Yaskawa INFORM job: KRIS7_V2.JBI

/JOB
//NAME KRIS7_V2
//POS
///NPOS 420,420,420,15,0,0
///TOOL 0
///POSTYPE PULSE
///PULSE
C00000=4302,-119221,-120806,-3568,29214,482
C00001=4302,-119221,-120806,-3568,29214,482
C00002=-36471,-76527,-106813,19264,71481,77238
C00003=-63812,-119516,-80644,-27282,71106,59809
C00004=-86670,-29465,-24103,-33182,93398,46515
C00005=-88663,-31189,-25266,-33292,92471,45985
C00006=-89600,-31952,-25776,-33339,92036,45737
C00007=-88663,-31189,-25266,-33292,92471,45985
C00008=-88663,-31929,-28188,-33361,93666,45629
C00009=-101397,-33118,-34088,-22474,91022,41668
C00010=-101397,-32934,-33069,-22469,90527,41762
C00011=-101397,-33275,-35023,-22483,91481,41581
C00012=-104499,20623,14787,-23283,115207,62973
C00013=-104352,17765,12486,-23220,115200,63034
C00014=-104529,15851,10717,-23303,115245,62949
C00015=-104352,17765,12486,-23220,115200,63034
C00016=-100086,19810,13187,-22516,115799,63398
C00017=-93288,781,-1160,-33549,91987,44264
C00018=-95103,1586,-482,-33591,91265,43744
C00019=-95638,1156,-842,-33600,91054,43591
C00020=-95103,1586,-482,-33591,91265,43744
C00021=-100253,-3614,-11898,-25466,91372,41970
C00022=-107199,-8537,-17665,-19004,89460,40114
C00023=-108350,-8919,-17473,-17740,88760,39873
C00024=-102096,-5783,-13006,-25389,90415,41488
C00025=-93175,-13453,-24658,-25770,96080,43586
C00026=-29596,-126908,-80456,-16683,91164,67663
C00027=-130966,-130992,-81417,14801,93022,-34731
C00028=-139735,-123676,-71676,23223,79574,-40827
C00029=-136755,-124231,-71804,23689,78586,-39979
C00030=-134984,-124514,-71869,23951,78010,-39473
C00031=-136755,-124231,-71804,23689,78586,-39979
C00032=-136306,-124758,-74432,23664,79703,-39597
C00033=-105195,-127447,-79852,15126,73259,-28242
C00034=-104798,-126140,-77647,15190,72530,-28198
C00035=-108375,-128078,-79564,15067,73342,-29336
C00036=-112121,-93277,-65445,16297,96104,-47809
C00037=-116095,-84503,-58814,18813,102506,-48434
C00038=-114391,-86924,-59797,19239,101506,-47972
C00039=-116095,-84503,-58814,18813,102506,-48434
C00040=-117812,-129995,-81150,14641,74986,-32390
C00041=-118791,-92886,-67151,14205,85296,-31516
C00042=-116748,-92781,-67110,14299,84968,-30842
C00043=-115499,-92681,-67072,14351,84774,-30431
C00044=-116748,-92781,-67110,14299,84968,-30842
C00045=-116748,-94243,-70296,14285,86141,-30707
C00046=-102870,-92009,-70676,9222,86435,-25689
C00047=-102870,-90997,-68303,9229,85506,-25758
C00048=-102870,-92009,-70676,9222,86435,-25689
C00049=-124106,-98193,-79828,8318,91183,-32632
C00050=-120990,-117719,-86799,1028,78019,83969
C00051=-103618,-122878,-84450,6731,45671,69045
C00052=-107839,-39273,-43881,11021,86771,60654
C00053=-102663,-26959,-34255,5037,90909,61236
C00054=-106417,-22492,-30421,10624,98396,60708
C00055=-103076,-37240,-40581,8849,97261,61678
C00056=-110992,-39766,-43585,17340,97602,59383
C00057=-111851,-103912,-94699,10334,87868,68255
C00058=-100525,-93554,-87313,9422,87254,72087
C00059=-95765,-72558,-76889,7644,100510,59309
C00060=-95463,-76426,-71939,16938,115118,61391
C00061=-102124,-64154,-61473,23072,122501,60539
C00062=-108072,-63754,-61449,27079,123073,58329
C00063=-126453,-110744,-88068,25157,96958,85114
C00064=-124535,-114305,-86499,25277,93833,85163
C00065=-121951,-112497,-85625,25654,93398,86032
C00066=-116232,-108405,-84002,26384,92604,88006
C00067=-122754,-106725,-87203,25770,97209,86568
C00068=-142865,-91008,-85242,17891,113758,73123
C00069=-142005,-90205,-84914,18160,113770,73464
C00070=-93871,-48257,-54590,-14207,101968,-48555
C00071=-106716,17042,-5346,-15024,102835,-53222
C00072=-114740,-14345,-34597,-13608,101053,-59815
C00073=-127078,-3386,-21930,-8482,103399,-53955
C00074=-129021,-1243,-17298,-7607,102543,-53064
C00075=-129893,-13096,-22178,-14005,113849,-54571
C00076=-129597,-5294,-13720,-15224,118044,-55057
C00077=-122058,-3228,-13278,-23261,119236,-52777
C00078=-102997,28917,14853,-20600,116287,-84527
C00079=-102792,-6395,-13177,-23260,105514,-87254
C00080=-105472,-3384,-9862,-23514,105257,-88219
C00081=-107060,-2107,-8876,-23770,104848,-88744
C00082=-104416,1445,-8009,-23523,106791,-88129
C00083=-100743,5943,-9423,-11985,113108,-51981
C00084=-104100,-22795,-28366,-25068,61310,-50210
C00085=-122112,-33809,-21710,-17217,45375,-58941
C00086=-130767,-31374,-20493,-827,48037,-55558
C00087=-127443,-25046,-15801,-6227,47707,-53970
C00088=-124818,-6385,-1356,-9028,48013,-52772
C00089=-117469,-7945,-6130,-22808,51414,-49873
C00090=-27812,-119319,-87277,-42007,83182,-24370
C00091=-5621,-139291,-109992,-39952,96377,80222
C00092=-5621,-139291,-109992,-39952,96377,80222
C00093=87039,-115654,-82424,8022,52039,63522
C00094=129513,-144814,-136934,9080,53426,64546
C00095=129513,-144814,-136934,9080,53426,64546
C00096=129513,-109632,-69732,14359,30578,61412
C00097=129513,-83278,-28536,22379,19314,57484
C00098=122399,-55102,-4999,-8402,35911,61097
C00099=119920,-45288,5620,-7331,30390,60229
C00100=119750,-46058,4611,-7150,30605,60108
C00101=119750,-45110,6218,-7257,30106,60163
C00102=119736,-46268,4531,-7151,30546,60106
C00103=119736,-47979,3777,-7238,30135,60151
C00104=119727,-46869,5444,-7329,29678,60198
C00105=119739,-46062,5830,-7299,29854,60181
C00106=119715,-47768,4014,-7231,30094,60141
C00107=122330,-55612,-6297,-8657,32618,61353
C00108=121709,-73745,-24049,9098,30676,53116
C00109=129398,-114812,-46545,3278,22913,57364
C00110=129398,-114812,-46545,3278,22913,57364
C00111=147189,-126166,-80752,5474,34460,60082
C00112=165214,-137669,-115409,7698,46160,62836
C00113=176409,-144814,-136934,9080,53426,64546
C00114=176409,-109327,-69248,14418,30440,61382
C00115=137996,-109327,-69248,14418,30440,61382
C00116=136854,5077,41656,21727,21645,57624
C00117=123203,14789,51546,53172,38991,40073
C00118=123077,34948,78392,59944,35543,36223
C00119=123077,37993,83408,61838,34770,35183
C00120=123098,35348,79007,60153,35442,36112
C00121=123139,31348,74887,59568,35673,36443
C00122=123149,34907,80133,61289,34946,35499
C00123=123130,37074,82445,61677,34805,35280
C00124=123183,30422,73312,58971,35912,36781
C00125=123599,57381,99984,51632,43856,40437
C00126=128629,59731,102899,52063,41097,41453
C00127=130023,30320,69348,52154,35987,38987
C00128=132104,19481,50493,23737,37003,47692
C00129=136200,48792,78585,9333,46433,53780
C00130=127667,43842,73216,11867,48213,50363
C00131=127110,36942,61073,12684,52130,50324
C00132=125174,17943,48073,21449,38985,45601
C00133=109988,7135,45797,56276,48109,34557
C00134=110783,-2370,26113,10588,43916,42309
C00135=96618,15106,36280,16308,48845,36588
C00136=99195,57631,83562,8929,54990,39222
C00137=83229,75338,108095,18392,45531,30732
C00138=82057,52050,70954,17595,54461,31693
C00139=99279,-29834,2408,12633,51480,38376
C00140=124602,-34297,-476,3581,48489,48797
C00141=129000,-155474,-110821,1722,53982,50766
C00142=129000,-186332,-136923,1718,54189,50769
C00143=129000,-186332,-136923,1718,54189,50769
C00144=124634,-42983,-17396,3288,54424,49011
C00145=119975,43106,65207,5416,48088,46799
C00146=124227,21838,45287,-4126,60993,49348
C00147=115102,22260,45694,-2630,60591,46004
C00148=111900,23179,46586,-2094,60423,44829
C00149=106599,25422,48781,-1196,60121,42879
C00150=109500,51617,73450,-2873,46958,44240
C00151=119708,-19564,1692,5024,54962,47046
C00152=124398,4257,31803,38326,49723,41965
C00153=124500,-5455,16693,36249,53145,43496
C00154=123978,22175,41893,32824,63757,46964
C00155=136633,26599,46213,31259,58773,50852
C00156=137127,47274,64261,33367,46328,47205
C00157=127043,-60461,-47717,31537,61680,47716
C00158=130427,-104246,-66216,34447,50964,45598
C00159=130427,-131180,-133049,27346,74705,52630
C00160=129293,-131648,-133187,27764,74930,52255
C00161=129293,-112975,-80869,32941,55210,46617
C00162=125224,-26758,-13299,33226,59088,46051
C00163=97492,-17863,6740,47317,62068,35221
C00164=76763,21057,43225,48272,71101,29312
C00165=80709,51150,75439,39481,73131,33496
C00166=101893,22474,45257,39781,66883,40263
C00167=98002,-1326,18556,46821,62661,35806
C00168=97492,-17863,6740,47317,62068,35221
C00169=125224,-26758,-13299,33226,59088,46051
C00170=129293,-131648,-133187,27764,74930,52255
C00171=129293,-130373,-135142,27565,76585,52657
C00172=129293,-130373,-135142,27565,76585,52657
C00173=129293,-130373,-135142,27565,76585,52657
C00174=126775,-65943,-41926,33631,56357,45828
C00175=146499,-5820,8509,-12483,47348,74367
C00176=133227,18598,33392,-5127,43166,68552
C00177=134087,40556,59352,-4333,44134,68757
C00178=109518,39473,58200,8432,44907,57480
C00179=110804,22133,33080,8574,45677,58038
C00180=95832,-100308,-60228,18401,42759,50383
C00181=85717,-180836,-128237,23276,45701,46095
C00182=134324,-194207,-130804,-6935,34984,69726
C00183=134324,-194207,-130804,-6935,34984,69726
C00184=134324,-194207,-130804,-6935,34984,69726
C00185=126554,-62104,-55568,-768,56192,65237
C00186=102691,-29899,-32559,11070,60126,55987
C00187=93699,-1684,15739,18283,46963,50224
C00188=95177,34388,59282,20423,38809,49091
C00189=95427,37375,44105,11480,58003,52927
C00190=82804,57701,66332,15963,56969,47713
C00191=80078,42075,52490,24500,50349,44630
C00192=92595,-4722,8571,18053,49920,50291
C00193=90890,13188,28851,45241,66990,53478
C00194=96516,51970,78121,48970,56932,51018
C00195=108766,35550,55769,36284,51974,56943
C00196=109501,48300,76470,39344,46724,54946
C00197=112089,47430,75488,38680,45769,55875
C00198=109461,35195,57508,36711,50675,56747
C00199=102961,43860,64049,37370,53600,54832
C00200=117347,37004,56694,33344,48695,60037
C00201=107165,27849,47408,45061,56134,56400
C00202=93699,-1684,15739,18283,46963,50224
C00203=126554,-62104,-55568,-768,56192,65237
C00204=132741,-190295,-136907,-5065,40605,68463
C00205=132741,-190295,-136907,-5065,40605,68463
C00206=132741,-190295,-136907,-5065,40605,68463
C00207=132741,-190295,-136907,-5065,40605,68463
C00208=126216,-48827,-32555,-652,48851,65144
C00209=116157,12397,26645,-836,43828,61032
C00210=107201,15073,29086,4732,43915,56787
C00211=108708,45240,59560,984,53519,57995
C00212=105889,47117,61614,1966,53270,56850
C00213=104117,15965,27840,6481,45345,55424
C00214=116157,12397,26645,-836,43828,61032
C00215=115184,32776,48658,-853,48273,60616
C00216=102009,39914,56094,5283,47719,54846
C00217=104295,38849,56164,-3583,45498,56420
C00218=106773,10666,21679,-1556,45201,57174
C00219=121513,8451,23347,32656,44981,60126
C00220=121479,33249,54130,32703,45073,60132
C00221=136244,38436,59676,26271,39414,66032
C00222=133358,13884,30500,26959,39421,64637
C00223=126216,-48827,-32555,-652,48851,65144
C00224=132741,-190295,-136907,-5065,40605,68463
C00225=132741,-190295,-136907,-5065,40605,68463
C00226=132741,-190295,-136907,-5065,40605,68463
C00227=132741,-190295,-136907,-5065,40605,68463
C00228=126554,-62104,-55568,-768,56192,65237
C00229=93699,-1684,15739,18283,46963,50224
C00230=109219,22842,33799,17593,55341,60017
C00231=114933,32716,55729,7970,41115,61622
C00232=98115,43367,67193,11592,40390,54327
C00233=92675,33947,50979,20393,49569,52577
C00234=113935,26100,44118,24451,47496,60162
C00235=114558,35388,59860,26260,42851,59091
C00236=117732,34768,59212,24806,41998,60459
C00237=114305,24559,43264,24398,47147,60243
C00238=99844,11402,27037,25299,53213,55440
C00239=126554,-62104,-55568,-768,56192,65237
C00240=132741,-190295,-136907,-5065,40605,68463
C00241=132741,-190295,-136907,-5065,40605,68463
C00242=132741,-190295,-136907,-5065,40605,68463
C00243=132741,-190295,-136907,-5065,40605,68463
C00244=126216,-48827,-32555,-652,48851,65144
C00245=134748,7082,18366,-200,46227,68791
C00246=132038,36511,51354,2924,49864,67481
C00247=110399,36003,50767,11764,51912,58463
C00248=101806,27679,40045,16592,51225,54569
C00249=102258,33237,49963,17192,48019,54198
C00250=104874,31614,48575,4374,45128,56525
C00251=106858,16986,29459,6761,48587,57166
C00252=113156,-2573,6178,11839,50347,59373
C00253=100847,-116604,-69788,21646,41420,51852
C00254=93537,-194381,-130385,26473,40988,47897
C00255=64846,-189571,-124664,-20885,48631,75512
C00256=85742,-187574,-126898,-2819,30744,64627
C00257=124193,-185785,-128899,13362,14722,54877
C00258=104459,-185785,-128899,13362,14722,54877
C00259=137185,-168918,-120422,-22616,31853,56508
C00260=103466,-143035,-89833,18127,44217,-664
C00261=153034,-42791,-3789,-574,51224,21077
C00262=154411,-23786,22188,6392,45845,11810
C00263=163692,-14831,30793,3045,43978,15753
C00264=162658,-12144,32796,3380,44162,15317
C00265=162658,-10372,35929,3443,43146,15280
C00266=162658,-10822,35136,3427,43403,15291
C00267=163644,-13399,33193,3102,43239,15709
C00268=163644,-12612,34572,3127,42795,15690
C00269=163043,-11060,35746,3327,42891,15434
C00270=163515,-12286,34819,3170,42815,15635
C00271=166152,-32133,5550,1997,50546,16952
C00272=100006,-46830,-3879,17345,57754,-8477
C00273=55652,-4276,24712,7053,56203,-22524
C00274=50070,19037,58848,16400,45172,-27179
C00275=51341,29328,71603,16783,42484,-27133
C00276=51341,32600,77102,17341,40853,-27469
C00277=51341,31422,75137,17137,41430,-27347
C00278=50264,28853,72458,17349,41942,-27728
C00279=50264,30492,75208,17635,41129,-27900
C00280=50738,31631,76404,17545,40896,-27733
C00281=50419,30858,75590,17605,41054,-27844
C00282=50419,14018,45638,14959,50461,-26136
C00283=53903,-12653,21571,13778,50962,-24612
C00284=66094,-67687,-18476,10677,45688,-20127
C00285=87454,-109874,-47340,-27972,40441,7116
C00286=78946,-55292,-6224,-23492,40558,2756
C00287=70027,-40972,10385,-20890,35738,-464
C00288=63439,-31094,22495,-18522,32104,-3061
C00289=63439,-29243,25592,-19018,31198,-2801
C00290=75556,-28394,37292,-62320,27769,16956
C00291=74155,-27422,37887,-61985,27131,16453
C00292=64318,-30449,24372,-21159,31089,-1672
C00293=67917,-25293,27676,-22824,32488,-51
C00294=67917,-25293,27676,-22824,32488,-51
C00295=68696,-24050,28500,-23162,32795,289
C00296=67917,-25293,27676,-22824,32488,-51
C00297=75368,-51805,-10970,-21451,43738,562
C00298=86139,-25078,5298,-24076,50017,4008
C00299=83917,-18337,16451,-24570,46284,3982
C00300=79836,-11066,25880,-23931,43276,2865
C00301=79836,-9413,28995,-24399,42297,3151
C00302=86314,-11086,32289,-42271,40319,10375
C00303=84998,-9998,33124,-41890,39785,9892
C00304=80963,-11349,26642,-26884,42529,4054
C00305=82363,-6834,30155,-27320,43093,4575
C00306=82761,-5465,31244,-27447,43243,4725
C00307=83186,-3958,32457,-27584,43396,4888
C00308=82761,-5465,31244,-27447,43243,4725
C00309=87385,-23200,183,-25112,53654,3858
C00310=88611,-6659,17671,-26227,51974,4862
C00311=85936,239,26154,-25964,49655,4281
C00312=85936,1480,28752,-26325,48787,4530
C00313=91127,630,32748,-40408,46738,9768
C00314=90313,1326,33333,-40211,46382,9497
C00315=86792,7,26768,-28149,49107,5083
C00316=90602,-33059,-4237,-28517,52203,5912
C00317=94576,-67258,-23025,57506,77870,-531
C00318=122383,-58832,-3556,65417,58097,774
C00319=127343,-13643,25366,63114,57669,4189
C00320=131296,13324,53885,65824,53660,3026
C00321=131296,14618,56173,66322,53341,2642
C00322=130824,14275,55697,67245,54004,2465
C00323=131723,14569,55971,67399,53464,2593
C00324=130860,14268,55674,67244,53987,2476
C00325=127124,-5804,29633,63377,58737,4694
C00326=126701,-15037,22522,63119,61223,3769
C00327=126701,1136,51385,68187,57095,-774
C00328=131284,6353,59362,70779,53649,-1335
C00329=131284,8754,63319,71617,53230,-1977
C00330=131284,6353,59362,70779,53649,-1335
C00331=132452,6685,59657,71098,52984,-1198
C00332=131284,6353,59362,70779,53649,-1335
C00333=131052,11501,64001,70861,53706,-1474
C00334=130893,14100,66417,70922,53742,-1574
C00335=130719,17099,69269,71021,53763,-1708
C00336=130893,14100,66417,70922,53742,-1574
C00337=128315,-22064,27147,66784,57381,941
C00338=129627,-37207,17556,68184,55855,186
C00339=130148,-23471,44300,74760,52317,-4741
C00340=135320,-14449,56479,79067,48853,-5949
C00341=135320,-12066,60154,79963,48630,-6563
C00342=135320,-14449,56479,79067,48853,-5949
C00343=137070,-14043,56767,79770,47945,-5809
C00344=135320,-14449,56479,79067,48853,-5949
C00345=134716,-10676,59212,78597,49226,-5841
C00346=134466,-8976,60486,78417,49378,-5807
C00347=134182,-6930,62050,78227,49545,-5776
C00348=134466,-8976,60486,78417,49378,-5807
C00349=106496,-51026,-9475,59829,73743,881
C00350=106496,-62277,-31108,58328,77765,3910
C00351=137468,-45448,-13164,23993,62707,9546
C00352=142031,-34381,-3630,18745,59946,9254
C00353=153480,-23481,18954,7895,48240,10284
C00354=154576,-15419,32985,7624,43640,10304
C00355=154522,-15140,33190,7639,43662,10282
C00356=163868,-10589,37972,6252,39486,12143
C00357=163705,-4288,45034,21073,38117,2051
C00358=163923,-2936,48273,26703,35302,170
C00359=146970,-27557,19782,29282,44621,-5055
C00360=77984,-28544,12598,9594,52255,-4511
C00361=87028,-14899,33509,-8097,43242,2023
C00362=86974,-14913,33498,-8080,43236,2001
C00363=77485,-7266,39372,-4959,42873,-2067
C00364=74579,-2521,47308,-17915,35684,548
C00365=75615,102,52227,-26296,32839,3633
C00366=84696,-19604,28451,-27180,39406,6073
C00367=87454,-109874,-47340,-27972,40441,7116
C00368=87454,-109874,-47340,-27972,40441,7116
C00369=73980,-36973,3355,-18473,60366,27525
C00370=58877,-27993,19766,-16405,50257,19650
C00371=71120,-6285,35203,-17245,53240,22132
C00372=69479,-8808,33067,-14788,50723,16894
C00373=73605,-31096,1389,-14177,59206,17320
C00374=72431,-18207,17991,-16956,51529,14828
C00375=73562,-15726,19761,-17396,52120,15565
C00376=83313,14185,44247,-21039,56473,22237
C00377=84211,-11070,13701,-18734,53182,26231
C00378=82998,-523,24465,-18637,51768,25979
C00379=82448,-570,28041,-15362,40529,26924
C00380=77134,-2165,39833,11119,14146,19838
C00381=76844,-12553,31864,7458,12108,20601
C00382=84341,-54767,463,-16268,10060,32559
C00383=79893,-46463,9240,-49361,8484,37720
C00384=71243,-22477,30789,30336,5200,-490
C00385=70979,-19028,33557,31433,5346,-1026
C00386=68683,-10375,50772,112552,4351,-37626
C00387=72976,-34040,25530,30096,2440,-170
C00388=51638,-47354,18402,88201,13764,-30312
C00389=50365,-30767,37744,101133,14655,-36527
C00390=46532,-17600,60099,119714,18815,-46088
C00391=50533,-52861,21550,106572,14840,-38992
C00392=66288,-93178,-46103,5866,60369,16168
C00393=112510,-98188,-44790,18471,62864,-44268
C00394=149625,-37879,6780,17046,57011,-35751
C00395=155605,-32525,16928,15112,50177,-29308
C00396=149418,-7594,34122,13784,51545,-27133
C00397=143716,-10385,36525,25765,46016,-27057
C00398=147766,-22217,9496,11268,57983,-23560
C00399=146875,-12758,20894,15319,55227,-24771
C00400=146053,-8471,24161,15451,55560,-25047
C00401=142035,19351,48051,16301,55907,-26583
C00402=141803,14161,44980,18392,51510,-21349
C00403=142040,5818,24378,13474,61789,-22474
C00404=138840,15265,37176,20739,58625,-24937
C00405=138706,17261,38894,20771,58629,-24991
C00406=139526,10572,40705,23596,37058,-29346
C00407=140566,11430,47120,26457,25355,-31911
C00408=140419,-8993,28489,25719,26277,-31573
C00409=142059,-17553,21658,25375,25949,-31323
C00410=143624,-11159,28730,24740,24544,-30775
C00411=144392,-5853,43056,31020,18891,-33660
C00412=150093,-42733,14524,24992,16002,-29807
C00413=146967,-32270,24662,40502,20136,-34953
C00414=144755,-20255,35089,33636,31779,-30408
C00415=144236,-61611,5153,41773,14596,-38681
C00416=136995,-150356,-85047,33892,64386,-36535
C00417=136995,-178339,-110283,33604,8697,-36217
C00418=130728,-161100,-136081,16173,33339,-28558
C00419=1271,-161100,-136081,16173,33339,-28558
BC00000=132383,679261,975760
BC00001=132383,679261,975760
BC00002=295325,674563,1075170
BC00003=396971,731967,797664
BC00004=396971,731967,797664
BC00005=396971,731967,797664
BC00006=396971,731967,797664
BC00007=396971,731967,797664
BC00008=396971,731967,797664
BC00009=396971,731967,797664
BC00010=396971,731967,797664
BC00011=396971,731967,797664
BC00012=396971,731967,797664
BC00013=396971,731967,797664
BC00014=396971,731967,797664
BC00015=396971,731967,797664
BC00016=396971,731967,797664
BC00017=396971,731967,797664
BC00018=396971,731967,797664
BC00019=396971,731967,797664
BC00020=396971,731967,797664
BC00021=396971,731967,797664
BC00022=396971,731967,797664
BC00023=396971,731967,797664
BC00024=396971,731967,797664
BC00025=396971,731967,797664
BC00026=396971,731967,797664
BC00027=1331,731967,797664
BC00028=1331,834817,797664
BC00029=1331,834817,797664
BC00030=1331,834817,797664
BC00031=1331,834817,797664
BC00032=1331,834817,797664
BC00033=1331,834817,797664
BC00034=1331,834817,797664
BC00035=1331,834817,797664
BC00036=1331,834817,797664
BC00037=1331,834817,797664
BC00038=1331,834817,797664
BC00039=1331,834817,797664
BC00040=1331,834817,797664
BC00041=1331,834817,797664
BC00042=1331,834817,797664
BC00043=1331,834817,797664
BC00044=1331,834817,797664
BC00045=1331,834817,797664
BC00046=1331,834817,797664
BC00047=1331,834817,797664
BC00048=1331,834817,797664
BC00049=1331,834817,797664
BC00050=1072,761065,516765
BC00051=1072,827865,516765
BC00052=1071,829671,517043
BC00053=1071,829895,517078
BC00054=1071,829895,517078
BC00055=1071,829895,517078
BC00056=1071,829895,517078
BC00057=768,829895,695080
BC00058=768,829895,695080
BC00059=768,829895,695080
BC00060=768,829895,695080
BC00061=768,829895,695080
BC00062=768,829895,695080
BC00063=768,829895,695080
BC00064=768,829895,695080
BC00065=768,829895,695080
BC00066=768,829895,695080
BC00067=768,829895,695080
BC00068=768,829895,695080
BC00069=768,686767,695080
BC00070=396971,681851,797664
BC00071=396971,731967,797664
BC00072=396971,731967,797664
BC00073=396971,731967,797664
BC00074=396971,731967,797664
BC00075=396971,731967,797664
BC00076=396971,731967,797664
BC00077=396971,731967,797664
BC00078=396971,731967,797664
BC00079=396971,731967,797664
BC00080=396971,731967,797664
BC00081=396971,731967,797664
BC00082=396971,731967,797664
BC00083=396971,731967,797664
BC00084=396971,731967,516765
BC00085=396971,731967,516765
BC00086=396971,731967,516765
BC00087=396972,731979,516765
BC00088=396971,731967,516765
BC00089=396971,731967,516765
BC00090=396971,731967,516765
BC00091=188286,731967,1013423
BC00092=188286,774486,1052805
BC00093=125948,1177450,1071719
BC00094=215453,1309115,984509
BC00095=345399,1357897,984509
BC00096=345399,1357897,984509
BC00097=345399,1230997,984509
BC00098=346767,1230997,984506
BC00099=346767,1230997,984506
BC00100=346767,1230997,984506
BC00101=346767,1230997,984506
BC00102=346767,1230997,984506
BC00103=346767,1230997,984506
BC00104=346767,1230997,984506
BC00105=346767,1230997,984506
BC00106=346767,1230997,984506
BC00107=346767,1230997,984506
BC00108=309515,1253158,984507
BC00109=309515,1253158,984507
BC00110=309515,1328360,1051553
BC00111=314470,1361455,1064018
BC00112=253389,1357693,1050986
BC00113=215453,1309115,984509
BC00114=215453,1309115,984509
BC00115=135997,1309115,984509
BC00116=135997,1309115,984509
BC00117=135997,1309115,984509
BC00118=135997,1309115,984505
BC00119=135997,1309115,984505
BC00120=135997,1309115,984505
BC00121=135997,1309115,984505
BC00122=135997,1309115,984505
BC00123=135997,1309115,984505
BC00124=135997,1309115,984505
BC00125=135997,1309115,984509
BC00126=135997,1309115,984509
BC00127=135997,1309115,984509
BC00128=135997,1309115,984509
BC00129=135997,1309115,984509
BC00130=135997,1309115,984509
BC00131=135997,1309115,984509
BC00132=135997,1309115,984509
BC00133=135997,1309115,984509
BC00134=135997,1309115,984509
BC00135=94463,1309115,955550
BC00136=94463,1309115,963176
BC00137=94463,1309115,963176
BC00138=94463,1309115,963176
BC00139=94463,1309115,963176
BC00140=141941,1309115,963176
BC00141=141941,1309115,963176
BC00142=223116,1330631,963176
BC00143=328548,1330631,963176
BC00144=328548,1330631,963176
BC00145=328548,1330631,963176
BC00146=328548,1285890,963176
BC00147=328548,1285890,963176
BC00148=328548,1285890,963176
BC00149=328548,1285890,963176
BC00150=328548,1330631,963176
BC00151=328548,1291307,959498
BC00152=328548,1293601,963176
BC00153=328548,1288886,905196
BC00154=328548,1288886,905196
BC00155=328548,1288886,905196
BC00156=328824,1330631,905196
BC00157=328824,1330631,905196
BC00158=328824,1330631,905196
BC00159=328824,1330631,905196
BC00160=151003,1330631,905196
BC00161=151003,1330631,905196
BC00162=151003,1330631,905196
BC00163=103648,1289163,905196
BC00164=103648,1289163,905196
BC00165=103648,1289163,905196
BC00166=103648,1289163,905196
BC00167=103648,1289163,905196
BC00168=103648,1289163,905196
BC00169=151003,1330631,905196
BC00170=151003,1330631,905196
BC00171=151003,1330631,905196
BC00172=303803,1330631,905196
BC00173=303803,1330631,763831
BC00174=303803,1330631,902112
BC00175=303803,1330631,902112
BC00176=303803,1330631,902112
BC00177=303803,1330631,902112
BC00178=303803,1330631,902112
BC00179=303803,1330631,902112
BC00180=303803,1330631,902112
BC00181=303803,1330631,1003127
BC00182=236612,1330631,1003127
BC00183=137483,1330631,1003127
BC00184=136337,1325904,719417
BC00185=136337,1325904,818715
BC00186=87820,1325904,842743
BC00187=87820,1325904,951848
BC00188=87820,1325904,951848
BC00189=87820,1320020,844218
BC00190=87820,1320020,844218
BC00191=87820,1325904,927335
BC00192=87820,1325904,927335
BC00193=87820,1325904,927335
BC00194=87820,1325904,927335
BC00195=87820,1325904,927335
BC00196=87820,1325904,927335
BC00197=87820,1325904,927335
BC00198=87820,1325904,927335
BC00199=87820,1325904,890762
BC00200=87820,1325904,890392
BC00201=87820,1325904,927335
BC00202=87820,1325904,951848
BC00203=136337,1325904,818715
BC00204=136337,1325904,818715
BC00205=136337,1325904,998300
BC00206=310720,1325904,998300
BC00207=310720,1325904,777065
BC00208=310720,1325904,891809
BC00209=310720,1325904,891809
BC00210=310720,1325904,891809
BC00211=310720,1325904,891809
BC00212=310720,1325904,891809
BC00213=310720,1325904,891809
BC00214=310720,1325904,891809
BC00215=310720,1325904,891809
BC00216=310720,1325904,891809
BC00217=310720,1325904,891809
BC00218=310720,1325904,891809
BC00219=310720,1325904,891809
BC00220=310720,1325904,891809
BC00221=310720,1325904,891809
BC00222=310720,1325904,891809
BC00223=310720,1325904,891809
BC00224=310720,1325904,777065
BC00225=310720,1325904,998300
BC00226=136337,1325904,998300
BC00227=136337,1325904,818715
BC00228=136337,1325904,818715
BC00229=87820,1325904,951848
BC00230=87820,1325904,927335
BC00231=87820,1325904,927335
BC00232=87820,1325904,927335
BC00233=87820,1325904,927335
BC00234=87820,1325904,927335
BC00235=87820,1325904,927335
BC00236=87820,1325904,927335
BC00237=87820,1325904,927335
BC00238=87820,1325904,927335
BC00239=136337,1325904,818715
BC00240=136337,1325904,818715
BC00241=136337,1325904,998300
BC00242=310720,1325904,998300
BC00243=310720,1325904,777065
BC00244=310720,1325904,891809
BC00245=310720,1325904,891809
BC00246=310720,1325904,891809
BC00247=310720,1325904,891809
BC00248=310720,1325904,891809
BC00249=310720,1325904,891809
BC00250=310720,1325904,891809
BC00251=310720,1325904,891809
BC00252=310720,1325904,891809
BC00253=310720,1325904,891809
BC00254=310720,1325904,1051225
BC00255=156074,1050332,1052018
BC00256=153940,1198656,1051600
BC00257=230237,1331507,1051225
BC00258=230237,1331507,1051225
BC00259=214487,1257960,1051225
BC00260=187930,1133951,1051225
BC00261=187930,1063861,1051225
BC00262=187930,1063861,1051225
BC00263=187931,1063862,1051199
BC00264=187931,1063862,1051199
BC00265=187931,1063862,1051199
BC00266=187931,1063862,1051199
BC00267=187931,1063862,1051199
BC00268=187931,1063862,1051199
BC00269=187931,1063862,1051199
BC00270=187931,1063862,1051199
BC00271=187931,1063862,1051199
BC00272=187930,1063861,1051225
BC00273=187930,1063861,1051225
BC00274=187930,1063861,1051225
BC00275=187930,1063861,1051225
BC00276=187930,1063861,1051225
BC00277=187930,1063861,1051225
BC00278=187930,1063861,1051225
BC00279=187930,1063861,1051225
BC00280=187930,1063861,1051225
BC00281=187930,1063861,1051225
BC00282=187930,1063861,1051225
BC00283=187930,1063861,1051225
BC00284=187930,1063861,1051225
BC00285=244084,1125149,1051225
BC00286=244084,1125149,1051225
BC00287=244084,1125149,1051225
BC00288=244084,1125149,1051225
BC00289=244084,1125149,1051225
BC00290=244084,1125149,1051225
BC00291=244084,1125149,1051225
BC00292=244084,1125149,1051225
BC00293=244084,1125149,1051225
BC00294=244084,1125149,1051225
BC00295=244084,1125149,1051225
BC00296=244084,1125149,1051225
BC00297=244084,1125149,1051225
BC00298=244084,1125149,1051225
BC00299=244084,1125149,1051225
BC00300=244084,1125149,1051225
BC00301=244084,1125149,1051225
BC00302=244084,1125149,1051225
BC00303=244084,1125149,1051225
BC00304=244084,1125149,1051225
BC00305=244084,1125149,1051225
BC00306=244084,1125149,1051225
BC00307=244084,1125149,1051225
BC00308=244084,1125149,1051225
BC00309=244084,1125149,1051225
BC00310=244084,1125149,1051225
BC00311=244083,1125149,1051222
BC00312=244083,1125149,1051222
BC00313=244083,1125149,1051222
BC00314=244083,1125149,1051222
BC00315=244083,1125149,1051222
BC00316=244083,1125149,1051222
BC00317=244083,1125148,1051219
BC00318=166173,1125148,1051219
BC00319=166173,1125148,1051219
BC00320=166173,1142192,1051219
BC00321=166173,1142192,1051219
BC00322=166173,1142192,1051219
BC00323=166173,1142192,1051219
BC00324=166173,1142192,1051219
BC00325=166173,1142192,1051219
BC00326=166173,1142192,1051219
BC00327=166173,1142192,1051219
BC00328=166173,1142192,1051219
BC00329=166173,1142192,1051219
BC00330=166173,1142192,1051219
BC00331=166173,1142192,1051219
BC00332=166173,1142192,1051219
BC00333=166173,1142192,1051219
BC00334=166173,1142192,1051219
BC00335=166173,1142192,1051219
BC00336=166173,1142192,1051219
BC00337=166173,1142192,1051219
BC00338=166173,1142192,1051219
BC00339=166173,1142192,1051219
BC00340=166173,1142192,1051219
BC00341=166173,1142192,1051219
BC00342=166173,1142192,1051219
BC00343=166173,1142192,1051219
BC00344=166173,1142192,1051219
BC00345=166173,1142192,1051219
BC00346=166173,1142192,1051219
BC00347=166173,1142192,1051219
BC00348=166173,1142192,1051219
BC00349=166173,1142192,1051219
BC00350=166173,1142192,1051219
BC00351=180177,1091773,1051223
BC00352=182943,1081815,1051224
BC00353=187709,1064658,1051225
BC00354=187930,1063861,1051225
BC00355=187930,1063861,1051225
BC00356=187930,1063861,1051225
BC00357=187930,1063861,1051225
BC00358=187930,1063861,1051225
BC00359=187930,1063861,1051225
BC00360=244084,1063861,1051225
BC00361=244084,1063861,1051225
BC00362=244084,1063861,1051225
BC00363=244084,1063861,1051225
BC00364=244084,1063861,1051225
BC00365=244084,1063861,1051225
BC00366=244084,1063861,1051225
BC00367=244084,1063861,1051225
BC00368=244084,1125149,1051225
BC00369=244084,1125149,1051225
BC00370=244084,1125149,1051225
BC00371=244084,1125149,1051225
BC00372=244084,1125149,1051225
BC00373=244084,1125149,1051225
BC00374=244084,1125149,1051225
BC00375=244084,1125149,1051225
BC00376=244084,1125149,1051225
BC00377=244084,1125149,1051225
BC00378=244084,1125149,1051225
BC00379=244084,1125149,1051225
BC00380=244084,1125149,1051225
BC00381=244084,1125149,1051225
BC00382=244084,1125149,1051225
BC00383=244084,1125149,1051225
BC00384=244084,1125149,1051225
BC00385=244084,1125149,1051222
BC00386=244084,1125149,1051225
BC00387=244084,1125149,1051225
BC00388=244084,1125149,1051225
BC00389=244083,1125149,1051223
BC00390=244084,1125149,1051225
BC00391=244084,1125149,1051225
BC00392=244084,1125149,1051225
BC00393=148492,1125149,1051225
BC00394=148492,1157650,1055882
BC00395=148492,1157650,1055882
BC00396=148492,1157650,1055882
BC00397=148493,1157650,1055879
BC00398=148492,1157650,1055882
BC00399=148492,1157650,1055882
BC00400=148492,1157650,1055882
BC00401=148492,1157650,1055882
BC00402=148492,1157650,1055882
BC00403=148492,1157650,1055882
BC00404=148492,1157650,1055882
BC00405=148492,1157650,1055882
BC00406=148492,1157650,1055881
BC00407=148492,1157650,1055882
BC00408=148492,1157650,1055882
BC00409=148492,1157650,1055882
BC00410=148492,1157650,1055882
BC00411=148492,1157650,1055882
BC00412=148492,1157650,1055882
BC00413=148492,1157650,1055882
BC00414=148492,1157650,1055882
BC00415=148492,1157650,1055882
BC00416=148492,1157650,1055882
BC00417=189366,1229859,1070827
BC00418=189366,1118575,1070827
BC00419=189366,734808,1070827
EC00000=443420,556475
EC00001=0,556475
EC00002=-88685,-556476
EC00003=-88685,-556476
EC00004=-88685,-556476
EC00005=-88685,-556476
EC00006=-88685,-556476
EC00007=-88685,-556476
EC00008=-88685,-556476
EC00009=-88685,-556476
EC00010=-88685,-556476
EC00011=-88685,-556476
EC00012=-88685,-556476
EC00013=-88685,-556476
EC00014=-88685,-556476
EC00015=-88685,-556476
EC00016=-88685,-556476
EC00017=-88685,-556476
EC00018=-88685,-556476
EC00019=-88685,-556476
EC00020=-88685,-556476
EC00021=-88685,-556476
EC00022=-88685,-556476
EC00023=-88685,-556476
EC00024=-88685,-556476
EC00025=-88685,-556476
EC00026=-88685,-556476
EC00027=-88685,-556476
EC00028=-88685,-556476
EC00029=-88685,-556476
EC00030=-88685,-556476
EC00031=-88685,-556476
EC00032=-88685,-556476
EC00033=-88685,-556476
EC00034=-88685,-556476
EC00035=-88685,-556476
EC00036=-88685,-556476
EC00037=-88685,-556476
EC00038=-88685,-556476
EC00039=-88685,-556476
EC00040=-88685,-556476
EC00041=-88685,-556476
EC00042=-88685,-556476
EC00043=-88685,-556476
EC00044=-88685,-556476
EC00045=-88685,-556476
EC00046=-88685,-556476
EC00047=-88685,-556476
EC00048=-88685,-556476
EC00049=-88685,-556476
EC00050=264893,-556476
EC00051=264893,-556476
EC00052=264346,-556476
EC00053=264278,-556476
EC00054=264278,-556476
EC00055=264278,-556476
EC00056=264278,-556476
EC00057=-85879,-556476
EC00058=-85879,-556476
EC00059=-85879,-556476
EC00060=-85879,-556476
EC00061=-85879,-556476
EC00062=-85879,-556476
EC00063=-85879,-556476
EC00064=-85879,-556476
EC00065=-85879,-556476
EC00066=-85879,-556476
EC00067=-85879,-556476
EC00068=-85879,-556476
EC00069=-85879,-556476
EC00070=-88685,-556476
EC00071=-88685,-556476
EC00072=-88685,-612042
EC00073=-88685,-612042
EC00074=-88685,-612042
EC00075=-88685,-612042
EC00076=-88685,-612042
EC00077=-88685,-612042
EC00078=-88685,-556476
EC00079=-88685,-556476
EC00080=-88685,-556476
EC00081=-88685,-556476
EC00082=-88685,-556476
EC00083=-88685,-556476
EC00084=264893,-556476
EC00085=264893,-605076
EC00086=264893,-605076
EC00087=264894,-605076
EC00088=264893,-605076
EC00089=264893,-605076
EC00090=264893,-556476
EC00091=264890,-556476
EC00092=264890,-556476
EC00093=-210078,-556477
EC00094=-270405,-556477
EC00095=-270405,-556477
EC00096=-270405,-556477
EC00097=-270405,-556477
EC00098=-270404,-556477
EC00099=-270404,-556477
EC00100=-270404,-556477
EC00101=-270404,-556477
EC00102=-270404,-556477
EC00103=-270404,-556477
EC00104=-270404,-556477
EC00105=-270404,-556477
EC00106=-270404,-556477
EC00107=-270404,-556477
EC00108=-270404,-556477
EC00109=-270404,-556477
EC00110=-270404,-556477
EC00111=-270404,-556477
EC00112=-270405,-556477
EC00113=-270405,-556477
EC00114=-270405,-556477
EC00115=-270405,-556477
EC00116=-270405,-556477
EC00117=-270405,-556477
EC00118=-270404,-556477
EC00119=-270404,-556477
EC00120=-270404,-556477
EC00121=-270404,-556477
EC00122=-270404,-556477
EC00123=-270404,-556477
EC00124=-270404,-556477
EC00125=-270405,-556477
EC00126=-270405,-556477
EC00127=-270405,-556477
EC00128=-270405,-556477
EC00129=-270405,-556477
EC00130=-270405,-556477
EC00131=-270405,-556477
EC00132=-270405,-556477
EC00133=-270405,-556477
EC00134=-270405,-556477
EC00135=-270405,-556477
EC00136=-270405,-556477
EC00137=-270405,-556477
EC00138=-270405,-556477
EC00139=-270405,-556477
EC00140=-270405,-556477
EC00141=-270405,-556477
EC00142=-270405,-556477
EC00143=-270405,-556477
EC00144=-270405,-556477
EC00145=-270405,-556477
EC00146=-270405,-556477
EC00147=-270405,-556477
EC00148=-270405,-556477
EC00149=-270405,-556477
EC00150=-270405,-556477
EC00151=-270405,-556477
EC00152=-270405,-556477
EC00153=-270405,-556477
EC00154=-270405,-556477
EC00155=-270405,-556477
EC00156=-270405,-556477
EC00157=-270405,-556477
EC00158=-270405,-556477
EC00159=-270405,-556477
EC00160=-270405,-556477
EC00161=-270405,-556477
EC00162=-270405,-556477
EC00163=-270405,-556477
EC00164=-270405,-556477
EC00165=-270405,-556477
EC00166=-270405,-556477
EC00167=-270405,-556477
EC00168=-270405,-556477
EC00169=-270405,-556477
EC00170=-270405,-556477
EC00171=-270405,-556477
EC00172=-270405,-556477
EC00173=-270405,-556477
EC00174=-270405,-556477
EC00175=-270405,-556477
EC00176=-270405,-556477
EC00177=-270405,-556477
EC00178=-270405,-556477
EC00179=-270405,-556477
EC00180=-270405,-556477
EC00181=-270405,-556477
EC00182=-270405,-556477
EC00183=-270405,-556477
EC00184=-270405,-556477
EC00185=-270405,-556477
EC00186=-270405,-556477
EC00187=-270405,-556477
EC00188=-270405,-556477
EC00189=-270405,-556477
EC00190=-270405,-556477
EC00191=-270405,-556477
EC00192=-270405,-556477
EC00193=-270405,-556477
EC00194=-270405,-556477
EC00195=-270405,-556477
EC00196=-270405,-556477
EC00197=-270405,-556477
EC00198=-270405,-556477
EC00199=-270405,-556477
EC00200=-270405,-556477
EC00201=-270405,-556477
EC00202=-270405,-556477
EC00203=-270405,-556477
EC00204=-270405,-556477
EC00205=-270405,-556477
EC00206=-270405,-556477
EC00207=-270405,-556477
EC00208=-270405,-556477
EC00209=-270405,-556477
EC00210=-270405,-556477
EC00211=-270405,-556477
EC00212=-270405,-556477
EC00213=-270405,-556477
EC00214=-270405,-556477
EC00215=-270405,-556477
EC00216=-270405,-556477
EC00217=-270405,-556477
EC00218=-270405,-556477
EC00219=-270405,-556477
EC00220=-270405,-556477
EC00221=-270405,-556477
EC00222=-270405,-556477
EC00223=-270405,-556477
EC00224=-270405,-556477
EC00225=-270405,-556477
EC00226=-270405,-556477
EC00227=-270405,-556477
EC00228=-270405,-556477
EC00229=-270405,-556477
EC00230=-270405,-556477
EC00231=-270405,-556477
EC00232=-270405,-556477
EC00233=-270405,-556477
EC00234=-270405,-556477
EC00235=-270405,-556477
EC00236=-270405,-556477
EC00237=-270405,-556477
EC00238=-270405,-556477
EC00239=-270405,-556477
EC00240=-270405,-556477
EC00241=-270405,-556477
EC00242=-270405,-556477
EC00243=-270405,-556477
EC00244=-270405,-556477
EC00245=-270405,-556477
EC00246=-270405,-556477
EC00247=-270405,-556477
EC00248=-270405,-556477
EC00249=-270405,-556477
EC00250=-270405,-556477
EC00251=-270405,-556477
EC00252=-270405,-556477
EC00253=-270405,-556477
EC00254=-270405,-556477
EC00255=-1607,-556476
EC00256=-143402,-556477
EC00257=-270405,-556477
EC00258=-270405,-556477
EC00259=-270405,-556477
EC00260=-270405,-556477
EC00261=-270405,-556477
EC00262=-270405,-556477
EC00263=-270402,-556478
EC00264=-270402,-556478
EC00265=-270402,-556478
EC00266=-270402,-556478
EC00267=-270402,-556478
EC00268=-270402,-556478
EC00269=-270402,-556478
EC00270=-270402,-556478
EC00271=-270402,-556478
EC00272=-270405,-556477
EC00273=-270405,-556477
EC00274=-270405,-556477
EC00275=-270405,-556477
EC00276=-270405,-556477
EC00277=-270405,-556477
EC00278=-270405,-556477
EC00279=-270405,-556477
EC00280=-270405,-556477
EC00281=-270405,-556477
EC00282=-270405,-556477
EC00283=-270405,-556477
EC00284=-270405,-556477
EC00285=-447795,-556477
EC00286=-447795,-556477
EC00287=-447795,-556477
EC00288=-447795,-556477
EC00289=-447795,-556477
EC00290=-447795,-556477
EC00291=-447795,-556477
EC00292=-447795,-556477
EC00293=-447795,-556477
EC00294=-447795,-556477
EC00295=-447795,-556477
EC00296=-447795,-556477
EC00297=-447795,-556477
EC00298=-447795,-556477
EC00299=-447795,-556477
EC00300=-447795,-556477
EC00301=-447795,-556477
EC00302=-447795,-556477
EC00303=-447795,-556477
EC00304=-447795,-556477
EC00305=-447795,-556477
EC00306=-447795,-556477
EC00307=-447795,-556477
EC00308=-447795,-556477
EC00309=-447795,-556477
EC00310=-447795,-556477
EC00311=-447793,-556477
EC00312=-447793,-556477
EC00313=-447793,-556477
EC00314=-447793,-556477
EC00315=-447793,-556477
EC00316=-447793,-556477
EC00317=-447791,-556477
EC00318=-447791,-556477
EC00319=-447791,-556477
EC00320=-447791,-556477
EC00321=-447791,-556477
EC00322=-447791,-556477
EC00323=-447791,-556477
EC00324=-447791,-556477
EC00325=-447791,-556477
EC00326=-447791,-556477
EC00327=-447791,-556477
EC00328=-447791,-556477
EC00329=-447791,-556477
EC00330=-447791,-556477
EC00331=-447791,-556477
EC00332=-447791,-556477
EC00333=-447791,-556477
EC00334=-447791,-556477
EC00335=-447791,-556477
EC00336=-447791,-556477
EC00337=-447791,-556477
EC00338=-447791,-556477
EC00339=-447791,-556477
EC00340=-447791,-556477
EC00341=-447791,-556477
EC00342=-447791,-556477
EC00343=-447791,-556477
EC00344=-447791,-556477
EC00345=-447791,-556477
EC00346=-447791,-556477
EC00347=-447791,-556477
EC00348=-447791,-556477
EC00349=-447791,-556477
EC00350=-447791,-556477
EC00351=-333615,-556477
EC00352=-311064,-556477
EC00353=-272209,-556477
EC00354=-270405,-556477
EC00355=-270405,-556477
EC00356=-270405,-556477
EC00357=-270405,-556477
EC00358=-270405,-556477
EC00359=-270405,-556477
EC00360=-270405,-556477
EC00361=-270405,-556477
EC00362=-270405,-556477
EC00363=-270405,-556477
EC00364=-270405,-556477
EC00365=-270405,-556477
EC00366=-270405,-556477
EC00367=-270405,-556477
EC00368=-447795,-556477
EC00369=-447795,-556477
EC00370=-447795,-556477
EC00371=-447795,-556477
EC00372=-447795,-556477
EC00373=-447795,-556477
EC00374=-447795,-556477
EC00375=-447795,-556477
EC00376=-447795,-556477
EC00377=-447795,-556477
EC00378=-447795,-556477
EC00379=-447795,-556477
EC00380=-447795,-556477
EC00381=-447795,-556477
EC00382=-447795,-556477
EC00383=-447795,-556477
EC00384=-447795,-556477
EC00385=-447794,-556477
EC00386=-447795,-556477
EC00387=-447795,-556477
EC00388=-447795,-556477
EC00389=-447794,-556478
EC00390=-447795,-556477
EC00391=-447795,-556477
EC00392=-447795,-556477
EC00393=-447795,-556477
EC00394=-447795,-556477
EC00395=-447795,-556477
EC00396=-447795,-556477
EC00397=-447793,-556477
EC00398=-447795,-556477
EC00399=-447795,-556477
EC00400=-447795,-556477
EC00401=-447795,-556477
EC00402=-447795,-556477
EC00403=-447795,-556477
EC00404=-447795,-556477
EC00405=-447795,-556477
EC00406=-447794,-556478
EC00407=-447795,-556477
EC00408=-447795,-556477
EC00409=-447795,-556477
EC00410=-447795,-556477
EC00411=-447795,-556477
EC00412=-447795,-556477
EC00413=-447795,-556477
EC00414=-447795,-556477
EC00415=-447795,-556477
EC00416=-447795,-556477
EC00417=-447795,-556477
EC00418=-71624,-556477
EC00419=15446,-556477
///POSTYPE BASE
///RECTAN
///RCONF 0,0,0,0,0,0,0,0,0,0,0,0,0,0,0,0,0,0,0,0,0,0,0,0
P00006=0.000,0.000,0.000,0.0000,0.0000,0.0000
P00032=1.957,0.503,-7.217,0.0000,0.0000,0.0000
///RCONF 0,0,0,0,1,0,0,0,0,0,0,0,0,0,0,0,0,0,0,0,0,0,0,0
P00033=-0.123,0.612,-5.012,0.0000,0.0000,0.0000
///RCONF 0,0,0,0,0,0,0,0,0,0,0,0,0,0,0,0,0,0,0,0,0,0,0,0
P00034=-0.304,0.773,-2.693,0.0000,0.0000,0.0000
P00035=2.817,0.591,-1.622,0.0000,0.0000,0.0000
P00040=-0.030,9.648,2.467,0.0000,0.0000,0.0000
P00041=0.192,3.924,0.305,0.0000,0.0000,0.0000
P00042=-0.217,1.941,0.413,0.0000,0.0000,0.0000
P00043=-0.044,-1.937,1.197,0.0000,0.0000,0.0000
P00044=0.687,-2.322,1.156,0.0000,0.0000,0.0000
P00045=-0.068,-0.810,1.603,0.0000,0.0000,0.0000
P00046=0.799,0.043,1.292,0.0000,0.0000,0.0000
P00048=2.411,0.025,-0.606,0.0000,0.0000,0.0000
P00049=3.413,-3.572,-1.618,0.0000,0.0000,0.0000
P00050=4.296,-4.501,-0.826,0.0000,0.0000,0.0000
//INST
///DATE 2025/03/14 12:45
///ATTR SC,RW
///GROUP1 RB1,BS1
///GROUP2 ST1
NOP
MOVJ C00000 BC00000 VJ=100.00  +MOVJ EC00000 VJ=100.00
MOVJ C00001 BC00001 VJ=100.00  +MOVJ EC00001 VJ=100.00
MOVJ C00002 BC00002 VJ=100.00  +MOVJ EC00002 VJ=100.00
CALL JOB:CLEAN-R1_KM_3P
MOVJ C00003 BC00003 VJ=100.00  +MOVJ EC00003 VJ=100.00
MOVJ C00004 BC00004 VJ=50.00  +MOVJ EC00004 VJ=50.00
SMOVL C00005 BC00005 V=83.3  +MOVJ EC00005
SREFP 3 C00006 BC00006  +REFP EC00006
CALL JOB:SEARCH-R1-S13D
SET P032 P006
SFTON3D P032
SMOVL C00007 BC00007 V=60.0  +MOVJ EC00007
SMOVL C00008 BC00008 V=133.3  +MOVJ EC00008
SMOVL C00009 BC00009 V=133.3  +MOVJ EC00009
SREFP 3 C00010 BC00010  +REFP EC00010
CALL JOB:SEARCH-R1-S13D
SET P032 P006
SFTON3D P032
SMOVL C00011 BC00011 V=60.0  +MOVJ EC00011
SMOVL C00012 BC00012 V=133.3  +MOVJ EC00012
SMOVL C00013 BC00013 V=133.3  +MOVJ EC00013
SREFP 3 C00014 BC00014  +REFP EC00014
CALL JOB:SEARCH-R1-S13D
SET P032 P006
SFTON3D P032
SFTOF3D
SMOVL C00015 BC00015 V=133.3  +MOVJ EC00015
SMOVL C00016 BC00016 V=200.0  +MOVJ EC00016
SFTOF3D
'S1
MOVJ C00017 BC00017 VJ=50.00  +MOVJ EC00017 VJ=50.00
'S2
SMOVL C00018 BC00018 V=60.0  +MOVJ EC00018
SREFP 3 C00019 BC00019  +REFP EC00019
CALL JOB:SEARCH-R1-S13D
SET P033 P006
SFTON3D P033
SMOVL C00020 BC00020 V=60.0  +MOVJ EC00020
SMOVL C00021 BC00021 V=133.3  +MOVJ EC00021
SMOVL C00022 BC00022 V=133.3  +MOVJ EC00022
SREFP 3 C00023 BC00023  +REFP EC00023
CALL JOB:SEARCH-R1-S13D
SET P033 P006
SFTON3D P033
SFTOF3D
SMOVL C00024 BC00024 V=83.3  +MOVJ EC00024
MOVJ C00025 BC00025 VJ=60.00  +MOVJ EC00025 VJ=60.00
MOVJ C00026 BC00026 VJ=60.00  +MOVJ EC00026 VJ=60.00
MOVJ C00027 BC00027 VJ=100.00  +MOVJ EC00027 VJ=60.00
MOVJ C00028 BC00028 VJ=60.00  +MOVJ EC00028 VJ=60.00
SMOVL C00029 BC00029 V=60.0  +MOVJ EC00029
SREFP 3 C00030 BC00030  +REFP EC00030
CALL JOB:SEARCH-R1-S13D
SET P034 P006
SFTON3D P034
SMOVL C00031 BC00031 V=60.0  +MOVJ EC00031
SMOVL C00032 BC00032 V=83.3  +MOVJ EC00032
SMOVL C00033 BC00033 V=83.3  +MOVJ EC00033
SREFP 3 C00034 BC00034  +REFP EC00034
CALL JOB:SEARCH-R1-S13D
SET P034 P006
SFTON3D P034
SMOVL C00035 BC00035 V=100.0  +MOVJ EC00035
SMOVL C00036 BC00036 V=133.3  +MOVJ EC00036
SMOVL C00037 BC00037 V=133.3  +MOVJ EC00037
SREFP 3 C00038 BC00038  +REFP EC00038
CALL JOB:SEARCH-R1-S13D
SET P034 P006
SFTON3D P034
SMOVL C00039 BC00039 V=133.3  +MOVJ EC00039
SMOVL C00040 BC00040 V=133.3  +MOVJ EC00040
SMOVL C00041 BC00041 V=250.0  +MOVJ EC00041
SMOVL C00042 BC00042 V=60.0  +MOVJ EC00042
SREFP 3 C00043 BC00043  +REFP EC00043
CALL JOB:SEARCH-R1-S13D
SET P035 P006
SFTON3D P035
SMOVL C00044 BC00044 V=60.0  +MOVJ EC00044
SMOVL C00045 BC00045 V=250.0  +MOVJ EC00045
SMOVL C00046 BC00046 V=250.0  +MOVJ EC00046
SREFP 3 C00047 BC00047  +REFP EC00047
CALL JOB:SEARCH-R1-S13D
SET P035 P006
SFTON3D P035
SMOVL C00048 BC00048 V=166.7  +MOVJ EC00048
SFTOF3D
MOVJ C00049 BC00049 VJ=30.00  +MOVJ EC00049 VJ=15.00
MOVJ C00050 BC00050 VJ=100.00  +MOVJ EC00050 VJ=50.00
MACRO1 MJ#(0) ARGF9
MOVJ C00051 BC00051 VJ=100.00  +MOVJ EC00051 VJ=15.00
SMOVL C00052 BC00052 V=666.7  +MOVJ EC00052
SFTON3D P035
SMOVL C00053 BC00053 V=166.7  +MOVJ EC00053
ARCON
SMOVL C00054 BC00054 V=6.7  +MOVJ EC00054
SMOVL C00055 BC00055 V=6.7  +MOVJ EC00055
ARCOF
TIMER T=1.00
SMOVL C00056 BC00056 V=166.7  +MOVJ EC00056
SFTOF3D
MOVJ C00057 BC00057 VJ=100.00  +MOVJ EC00057 VJ=100.00
MOVJ C00058 BC00058 VJ=15.00  +MOVJ EC00058 VJ=100.00
SFTON3D P035
SMOVL C00059 BC00059 V=166.7  +MOVJ EC00059
ARCON
SFTON3D P034
SMOVL C00060 BC00060 V=8.3  +MOVJ EC00060
SMOVL C00061 BC00061 V=8.3  +MOVJ EC00061
ARCOF
SMOVL C00062 BC00062 V=166.7  +MOVJ EC00062
SMOVL C00063 BC00063 V=500.0  +MOVJ EC00063
SMOVL C00064 BC00064 V=166.7  +MOVJ EC00064
ARCON
SMOVL C00065 BC00065 V=7.5  +MOVJ EC00065
SMOVL C00066 BC00066 V=7.5  +MOVJ EC00066
ARCOF
SFTOF3D
MOVJ C00067 BC00067 VJ=30.00  +MOVJ EC00067 VJ=60.00
MOVJ C00068 BC00068 VJ=100.00  +MOVJ EC00068 VJ=50.00
MOVJ C00069 BC00069 VJ=100.00  +MOVJ EC00069 VJ=15.00
MOVJ C00070 BC00070 VJ=100.00  +MOVJ EC00070 VJ=100.00
MOVJ C00071 BC00071 VJ=50.00  +MOVJ EC00071 VJ=50.00
SFTOF3D
MOVJ C00072 BC00072 VJ=100.00  +MOVJ EC00072 VJ=100.00
MOVJ C00073 BC00073 VJ=100.00  +MOVJ EC00073 VJ=100.00
SFTON3D P033
SMOVL C00074 BC00074 V=166.7  +MOVJ EC00074
ARCON
SFTON3D P032
SMOVL C00075 BC00075 V=8.3  +MOVJ EC00075
SMOVL C00076 BC00076 V=8.3  +MOVJ EC00076
ARCOF
SMOVL C00077 BC00077 V=166.7  +MOVJ EC00077
SMOVL C00078 BC00078 V=666.7  +MOVJ EC00078
SMOVL C00079 BC00079 V=133.3  +MOVJ EC00079
ARCON
SMOVL C00080 BC00080 V=7.5  +MOVJ EC00080
SMOVL C00081 BC00081 V=7.5  +MOVJ EC00081
ARCOF
SFTOF3D
SMOVL C00082 BC00082 V=133.3  +MOVJ EC00082
MOVJ C00083 BC00083 VJ=50.00  +MOVJ EC00083 VJ=50.00
MOVJ C00084 BC00084 VJ=100.00  +MOVJ EC00084 VJ=100.00
MOVJ C00085 BC00085 VJ=100.00  +MOVJ EC00085 VJ=100.00
SFTON3D P033
SMOVL C00086 BC00086 V=133.3  +MOVJ EC00086
ARCON
SMOVL C00087 BC00087 V=7.5  +MOVJ EC00087
ARCON
SMOVL C00088 BC00088 V=7.5  +MOVJ EC00088
ARCOF
MOVJ C00089 BC00089 VJ=50.00  +MOVJ EC00089 VJ=50.00
MOVJ C00090 BC00090 VJ=100.00  +MOVJ EC00090 VJ=100.00
CALL JOB:CLEAN-R1_KM_3P
MOVJ C00091 BC00091 VJ=100.00  +MOVJ EC00091 VJ=100.00
MOVJ C00092 BC00092 VJ=100.00  +MOVJ EC00092 VJ=100.00
COMM MOVJ C00093 BC00093 VJ=100.00  +MOVJ EC00093 VJ=100.00
COMM MOVJ C00094 BC00094 VJ=100.00  +MOVJ EC00094 VJ=50.00
COMM MOVJ C00095 BC00095 VJ=100.00  +MOVJ EC00095 VJ=50.00
COMM MOVJ C00096 BC00096 VJ=100.00  +MOVJ EC00096 VJ=50.00
COMM MOVJ C00097 BC00097 VJ=100.00  +MOVJ EC00097 VJ=50.00
COMM MOVJ C00098 BC00098 VJ=100.00  +MOVJ EC00098 VJ=15.00
COMM SFTOF3D
COMM MOVJ C00099 BC00099 VJ=15.00  +MOVJ EC00099 VJ=15.00
COMM SMOVL C00100 BC00100 V=100.0  +MOVJ EC00100
COMM SREFP 3 C00101 BC00101  +REFP EC00101
COMM CALL JOB:SEARCH-R1-S13D
COMM SET P041 P006
COMM SFTON3D P041
COMM SMOVL C00102 BC00102 V=100.0  +MOVJ EC00102
COMM SMOVL C00103 BC00103 V=83.3  +MOVJ EC00103
COMM SMOVL C00104 BC00104 V=83.3  +MOVJ EC00104
COMM SREFP 3 C00105 BC00105  +REFP EC00105
COMM CALL JOB:SEARCH-R1-S13D
COMM SET P041 P006
COMM SFTON3D P041
COMM SMOVL C00106 BC00106 V=100.0  +MOVJ EC00106
COMM SFTOF3D
COMM MOVJ C00107 BC00107 VJ=40.00  +MOVJ EC00107 VJ=100.00
COMM MOVJ C00108 BC00108 VJ=100.00  +MOVJ EC00108 VJ=15.00
COMM MOVJ C00109 BC00109 VJ=100.00  +MOVJ EC00109 VJ=15.00
COMM MOVJ C00110 BC00110 VJ=100.00  +MOVJ EC00110 VJ=15.00
COMM MOVJ C00111 BC00111 VJ=100.00  +MOVJ EC00111 VJ=15.00
COMM MOVJ C00112 BC00112 VJ=30.00  +MOVJ EC00112 VJ=15.00
COMM MOVJ C00113 BC00113 VJ=100.00  +MOVJ EC00113 VJ=50.00
COMM MOVJ C00114 BC00114 VJ=50.00  +MOVJ EC00114 VJ=50.00
COMM MOVJ C00115 BC00115 VJ=50.00  +MOVJ EC00115 VJ=50.00
COMM MOVJ C00116 BC00116 VJ=50.00  +MOVJ EC00116 VJ=50.00
COMM MOVJ C00117 BC00117 VJ=50.00  +MOVJ EC00117 VJ=50.00
COMM SFTOF3D
COMM SMOVL C00118 BC00118 V=83.3  +MOVJ EC00118
COMM SREFP 3 C00119 BC00119  +REFP EC00119
COMM CALL JOB:SEARCH-R1-S13D
COMM SET P040 P006
COMM SFTON3D P040
COMM SMOVL C00120 BC00120 V=100.0  +MOVJ EC00120
COMM SMOVL C00121 BC00121 V=133.3  +MOVJ EC00121
COMM SMOVL C00122 BC00122 V=83.3 PL=0  +MOVJ EC00122
COMM SREFP 3 C00123 BC00123  +REFP EC00123
COMM CALL JOB:SEARCH-R1-S13D
COMM SET P040 P006
COMM SFTON3D P040
COMM SMOVL C00124 BC00124 V=100.0  +MOVJ EC00124
COMM SFTOF3D
COMM MACRO1 MJ#(0) ARGF9
COMM SFTON3D P040
COMM SMOVL C00125 BC00125 V=133.3  +MOVJ EC00125
COMM ARCON
COMM SMOVL C00126 BC00126 V=11.7  +MOVJ EC00126
COMM ARCOF
COMM MOVJ C00127 BC00127 VJ=20.00  +MOVJ EC00127 VJ=15.00
COMM MOVJ C00128 BC00128 VJ=30.00  +MOVJ EC00128 VJ=15.00
COMM 'SPAWDZIC CZY SPOINA TRAFIA
COMM SMOVL C00129 BC00129 V=166.7  +MOVJ EC00129
COMM ARCON
COMM SMOVL C00130 BC00130 V=12.5  +MOVJ EC00130
COMM ARCOF
COMM SMOVL C00131 BC00131 V=333.3  +MOVJ EC00131
COMM MOVJ C00132 BC00132 VJ=50.00  +MOVJ EC00132 VJ=50.00
COMM MOVJ C00133 BC00133 VJ=100.00  +MOVJ EC00133 VJ=50.00
COMM MOVJ C00134 BC00134 VJ=100.00  +MOVJ EC00134 VJ=50.00
COMM MOVJ C00135 BC00135 VJ=100.00  +MOVJ EC00135 VJ=50.00
COMM SFTON3D P040
COMM SMOVL C00136 BC00136 V=250.0  +MOVJ EC00136
COMM ARCON
COMM SMOVL C00137 BC00137 V=11.7  +MOVJ EC00137
COMM ARCOF
COMM SFTOF3D
COMM MOVJ C00138 BC00138 VJ=25.00  +MOVJ EC00138 VJ=50.00
COMM MOVJ C00139 BC00139 VJ=100.00  +MOVJ EC00139 VJ=50.00
COMM MOVJ C00140 BC00140 VJ=100.00  +MOVJ EC00140 VJ=50.00
COMM MOVJ C00141 BC00141 VJ=100.00  +MOVJ EC00141 VJ=50.00
COMM MOVJ C00142 BC00142 VJ=100.00  +MOVJ EC00142 VJ=50.00
COMM MOVJ C00143 BC00143 VJ=100.00  +MOVJ EC00143 VJ=50.00
COMM SFTOF3D
COMM MOVJ C00144 BC00144 VJ=100.00  +MOVJ EC00144 VJ=50.00
COMM SFTOF3D
COMM MOVJ C00145 BC00145 VJ=100.00  +MOVJ EC00145 VJ=50.00
COMM SFTON3D P041
COMM SMOVL C00146 BC00146 V=200.0  +MOVJ EC00146
COMM ARCON
COMM SMOVL C00147 BC00147 V=10.8  +MOVJ EC00147
COMM ARCOF
COMM SMOVL C00148 BC00148 V=83.3  +MOVJ EC00148
COMM ARCON
COMM SMOVL C00149 BC00149 V=10.0  +MOVJ EC00149
COMM ARCOF
COMM SMOVL C00150 BC00150 V=250.0  +MOVJ EC00150
COMM MOVJ C00151 BC00151 VJ=50.00  +MOVJ EC00151 VJ=50.00
COMM MOVJ C00152 BC00152 VJ=15.00  +MOVJ EC00152 VJ=50.00
COMM SMOVL C00153 BC00153 V=250.0  +MOVJ EC00153
COMM MACRO1 MJ#(0) ARGF9
COMM SMOVL C00154 BC00154 V=200.0  +MOVJ EC00154
COMM ARCON
COMM SMOVL C00155 BC00155 V=11.7  +MOVJ EC00155
COMM ARCOF
COMM SMOVL C00156 BC00156 V=333.3  +MOVJ EC00156
COMM SFTOF3D
COMM MOVJ C00157 BC00157 VJ=100.00  +MOVJ EC00157 VJ=50.00
COMM MOVJ C00158 BC00158 VJ=100.00  +MOVJ EC00158 VJ=50.00
COMM MOVJ C00159 BC00159 VJ=100.00  +MOVJ EC00159 VJ=50.00
COMM MOVJ C00160 BC00160 VJ=100.00  +MOVJ EC00160 VJ=50.00
COMM MOVJ C00161 BC00161 VJ=100.00  +MOVJ EC00161 VJ=50.00
COMM MOVJ C00162 BC00162 VJ=100.00  +MOVJ EC00162 VJ=50.00
COMM MOVJ C00163 BC00163 VJ=100.00  +MOVJ EC00163 VJ=50.00
COMM MOVJ C00164 BC00164 VJ=20.00  +MOVJ EC00164 VJ=50.00
COMM SFTON3D P040
COMM SMOVL C00165 BC00165 V=83.3  +MOVJ EC00165
COMM ARCON
COMM SMOVL C00166 BC00166 V=11.7  +MOVJ EC00166
COMM ARCOF
COMM SMOVL C00167 BC00167 V=133.3  +MOVJ EC00167
COMM SFTOF3D
COMM MOVJ C00168 BC00168 VJ=50.00  +MOVJ EC00168 VJ=50.00
COMM MOVJ C00169 BC00169 VJ=100.00  +MOVJ EC00169 VJ=50.00
COMM MOVJ C00170 BC00170 VJ=100.00  +MOVJ EC00170 VJ=50.00
COMM MOVJ C00171 BC00171 VJ=100.00  +MOVJ EC00171 VJ=50.00
COMM MOVJ C00172 BC00172 VJ=100.00  +MOVJ EC00172 VJ=50.00
COMM MOVJ C00173 BC00173 VJ=100.00  +MOVJ EC00173 VJ=50.00
COMM MOVJ C00174 BC00174 VJ=100.00  +MOVJ EC00174 VJ=50.00
COMM MOVJ C00175 BC00175 VJ=100.00  +MOVJ EC00175 VJ=50.00
COMM MOVJ C00176 BC00176 VJ=15.00  +MOVJ EC00176 VJ=50.00
COMM SFTON3D P041
COMM SMOVL C00177 BC00177 V=133.3  +MOVJ EC00177
COMM ARCON
COMM SMOVL C00178 BC00178 V=11.7  +MOVJ EC00178
COMM ARCOF
COMM SMOVL C00179 BC00179 V=133.3  +MOVJ EC00179
COMM SFTOF3D
COMM MOVJ C00180 BC00180 VJ=100.00  +MOVJ EC00180 VJ=50.00
COMM MOVJ C00181 BC00181 VJ=100.00  +MOVJ EC00181 VJ=50.00
COMM MOVJ C00182 BC00182 VJ=100.00  +MOVJ EC00182 VJ=50.00
COMM MOVJ C00183 BC00183 VJ=100.00  +MOVJ EC00183 VJ=50.00
COMM MOVJ C00184 BC00184 VJ=100.00  +MOVJ EC00184 VJ=50.00
COMM MOVJ C00185 BC00185 VJ=100.00  +MOVJ EC00185 VJ=50.00
COMM MOVJ C00186 BC00186 VJ=100.00  +MOVJ EC00186 VJ=50.00
COMM MOVJ C00187 BC00187 VJ=100.00  +MOVJ EC00187 VJ=50.00
COMM MOVJ C00188 BC00188 VJ=15.00  +MOVJ EC00188 VJ=50.00
COMM SFTON3D P040
COMM SMOVL C00189 BC00189 V=133.3  +MOVJ EC00189
COMM ARCON
COMM SMOVL C00190 BC00190 V=11.7  +MOVJ EC00190
COMM ARCOF
COMM SMOVL C00191 BC00191 V=133.3  +MOVJ EC00191
COMM MOVJ C00192 BC00192 VJ=100.00  +MOVJ EC00192 VJ=50.00
COMM MOVJ C00193 BC00193 VJ=100.00  +MOVJ EC00193 VJ=50.00
COMM MOVJ C00194 BC00194 VJ=100.00  +MOVJ EC00194 VJ=50.00
COMM MOVJ C00195 BC00195 VJ=15.00  +MOVJ EC00195 VJ=15.00
COMM SMOVL C00196 BC00196 V=133.3  +MOVJ EC00196
COMM ARCON
COMM SMOVL C00197 BC00197 V=11.7  +MOVJ EC00197
COMM ARCOF
COMM SMOVL C00198 BC00198 V=133.3  +MOVJ EC00198
COMM SMOVL C00199 BC00199 V=133.3  +MOVJ EC00199
COMM ARCON
COMM SMOVL C00200 BC00200 V=11.7  +MOVJ EC00200
COMM ARCOF
COMM SFTOF3D
COMM SMOVL C00201 BC00201 V=133.3  +MOVJ EC00201
COMM MOVJ C00202 BC00202 VJ=100.00  +MOVJ EC00202 VJ=50.00
COMM MOVJ C00203 BC00203 VJ=100.00  +MOVJ EC00203 VJ=50.00
COMM MOVJ C00204 BC00204 VJ=100.00  +MOVJ EC00204 VJ=50.00
COMM MOVJ C00205 BC00205 VJ=100.00  +MOVJ EC00205 VJ=50.00
COMM MOVJ C00206 BC00206 VJ=100.00  +MOVJ EC00206 VJ=50.00
COMM MOVJ C00207 BC00207 VJ=100.00  +MOVJ EC00207 VJ=50.00
COMM MOVJ C00208 BC00208 VJ=100.00  +MOVJ EC00208 VJ=50.00
COMM MOVJ C00209 BC00209 VJ=100.00  +MOVJ EC00209 VJ=50.00
COMM MOVJ C00210 BC00210 VJ=50.00  +MOVJ EC00210 VJ=50.00
COMM SFTON3D P041
COMM SMOVL C00211 BC00211 V=16.7  +MOVJ EC00211
COMM ARCON
COMM SMOVL C00212 BC00212 V=8.3  +MOVJ EC00212
COMM ARCOF
COMM SMOVL C00213 BC00213 V=250.0  +MOVJ EC00213
COMM MOVJ C00214 BC00214 VJ=100.00  +MOVJ EC00214 VJ=50.00
COMM MACRO1 MJ#(0) ARGF9
COMM SMOVL C00215 BC00215 V=250.0  +MOVJ EC00215
COMM ARCON
COMM SMOVL C00216 BC00216 V=11.7  +MOVJ EC00216
COMM SMOVL C00217 BC00217 V=11.7  +MOVJ EC00217
COMM ARCOF
COMM SMOVL C00218 BC00218 V=166.7  +MOVJ EC00218
COMM SMOVL C00219 BC00219 V=666.7  +MOVJ EC00219
COMM SMOVL C00220 BC00220 V=250.0  +MOVJ EC00220
COMM ARCON
COMM SMOVL C00221 BC00221 V=11.7  +MOVJ EC00221
COMM ARCOF
COMM SFTOF3D
COMM SMOVL C00222 BC00222 V=166.7  +MOVJ EC00222
COMM MOVJ C00223 BC00223 VJ=100.00  +MOVJ EC00223 VJ=50.00
COMM MOVJ C00224 BC00224 VJ=100.00  +MOVJ EC00224 VJ=50.00
COMM MOVJ C00225 BC00225 VJ=100.00  +MOVJ EC00225 VJ=50.00
COMM MOVJ C00226 BC00226 VJ=100.00  +MOVJ EC00226 VJ=50.00
COMM MOVJ C00227 BC00227 VJ=100.00  +MOVJ EC00227 VJ=50.00
COMM MOVJ C00228 BC00228 VJ=50.00  +MOVJ EC00228 VJ=50.00
COMM MOVJ C00229 BC00229 VJ=50.00  +MOVJ EC00229 VJ=50.00
COMM MOVJ C00230 BC00230 VJ=50.00  +MOVJ EC00230 VJ=50.00
COMM SFTON3D P040
COMM SMOVL C00231 BC00231 V=166.7  +MOVJ EC00231
COMM ARCON
COMM SMOVL C00232 BC00232 V=11.7  +MOVJ EC00232
COMM ARCOF
COMM SMOVL C00233 BC00233 V=333.3  +MOVJ EC00233
COMM SMOVL C00234 BC00234 V=666.7  +MOVJ EC00234
COMM SMOVL C00235 BC00235 V=166.7  +MOVJ EC00235
COMM ARCON
COMM SMOVL C00236 BC00236 V=11.7  +MOVJ EC00236
COMM ARCOF
COMM SMOVL C00237 BC00237 V=333.3  +MOVJ EC00237
COMM SFTOF3D
COMM MOVJ C00238 BC00238 VJ=50.00  +MOVJ EC00238 VJ=50.00
COMM MOVJ C00239 BC00239 VJ=50.00  +MOVJ EC00239 VJ=50.00
COMM MOVJ C00240 BC00240 VJ=50.00  +MOVJ EC00240 VJ=50.00
COMM MOVJ C00241 BC00241 VJ=50.00  +MOVJ EC00241 VJ=50.00
COMM MOVJ C00242 BC00242 VJ=50.00  +MOVJ EC00242 VJ=50.00
COMM MOVJ C00243 BC00243 VJ=100.00  +MOVJ EC00243 VJ=50.00
COMM MOVJ C00244 BC00244 VJ=100.00  +MOVJ EC00244 VJ=50.00
COMM MOVJ C00245 BC00245 VJ=50.00  +MOVJ EC00245 VJ=50.00
COMM SFTON3D P041
COMM SMOVL C00246 BC00246 V=250.0  +MOVJ EC00246
COMM ARCON
COMM SMOVL C00247 BC00247 V=11.7  +MOVJ EC00247
COMM ARCOF
COMM SMOVL C00248 BC00248 V=250.0  +MOVJ EC00248
COMM SMOVL C00249 BC00249 V=250.0  +MOVJ EC00249
COMM ARCON
COMM SMOVL C00250 BC00250 V=10.8  +MOVJ EC00250
COMM ARCOF
COMM SMOVL C00251 BC00251 V=250.0  +MOVJ EC00251
COMM SMOVL C00252 BC00252 V=666.7  +MOVJ EC00252
COMM MOVJ C00253 BC00253 VJ=100.00  +MOVJ EC00253 VJ=50.00
COMM SSFTOF
COMM MOVJ C00254 BC00254 VJ=100.00  +MOVJ EC00254 VJ=50.00
COMM CALL JOB:CLEAN-R1_KM2
MOVJ C00255 BC00255 VJ=100.00  +MOVJ EC00255 VJ=100.00
MOVJ C00256 BC00256 VJ=100.00  +MOVJ EC00256 VJ=100.00
MOVJ C00257 BC00257 VJ=100.00  +MOVJ EC00257 VJ=100.00
MOVJ C00258 BC00258 VJ=100.00  +MOVJ EC00258 VJ=50.00
MOVJ C00259 BC00259 VJ=100.00  +MOVJ EC00259 VJ=15.00
MOVJ C00260 BC00260 VJ=100.00  +MOVJ EC00260 VJ=50.00
MOVJ C00261 BC00261 VJ=100.00  +MOVJ EC00261 VJ=50.00
MOVJ C00262 BC00262 VJ=15.00  +MOVJ EC00262 VJ=15.00
MOVJ C00263 BC00263 VJ=15.00  +MOVJ EC00263 VJ=50.00
SMOVL C00264 BC00264 V=83.3  +MOVJ EC00264
SREFP 3 C00265 BC00265  +REFP EC00265
CALL JOB:SEARCH-R1-S13D
SET P042 P006
SFTON3D P042
SMOVL C00266 BC00266 V=60.0  +MOVJ EC00266
SMOVL C00267 BC00267 V=133.3  +MOVJ EC00267
SMOVL C00268 BC00268 V=133.3  +MOVJ EC00268
SREFP 3 C00269 BC00269  +REFP EC00269
CALL JOB:SEARCH-R1-S13D
SET P042 P006
SFTON3D P042
SMOVL C00270 BC00270 V=60.0  +MOVJ EC00270
SFTOF3D
MOVJ C00271 BC00271 VJ=15.00  +MOVJ EC00271 VJ=15.00
MOVJ C00272 BC00272 VJ=15.00  +MOVJ EC00272 VJ=15.00
MOVJ C00273 BC00273 VJ=15.00  +MOVJ EC00273 VJ=15.00
MOVJ C00274 BC00274 VJ=15.00  +MOVJ EC00274 VJ=15.00
SMOVL C00275 BC00275 V=83.3  +MOVJ EC00275
SREFP 3 C00276 BC00276  +REFP EC00276
CALL JOB:SEARCH-R1-S13D
SET P043 P006
SFTON3D P043
SMOVL C00277 BC00277 V=60.0  +MOVJ EC00277
SMOVL C00278 BC00278 V=133.3  +MOVJ EC00278
SMOVL C00279 BC00279 V=133.3  +MOVJ EC00279
SREFP 3 C00280 BC00280  +REFP EC00280
CALL JOB:SEARCH-R1-S13D
SET P043 P006
SFTON3D P043
SMOVL C00281 BC00281 V=60.0  +MOVJ EC00281
MOVJ C00282 BC00282 VJ=30.00  +MOVJ EC00282 VJ=30.00
SFTOF3D
MOVJ C00283 BC00283 VJ=30.00  +MOVJ EC00283 VJ=30.00
MOVJ C00284 BC00284 VJ=30.00  +MOVJ EC00284 VJ=30.00
MOVJ C00285 BC00285 VJ=50.00  +MOVJ EC00285 VJ=50.00
MOVJ C00286 BC00286 VJ=50.00  +MOVJ EC00286 VJ=50.00
SFTOF3D
MOVJ C00287 BC00287 VJ=30.00  +MOVJ EC00287 VJ=30.00
SMOVL C00288 BC00288 V=83.3  +MOVJ EC00288
SREFP 3 C00289 BC00289  +REFP EC00289
CALL JOB:SEARCH-R1-S13D
SET P044 P006
SFTON3D P044
SMOVL C00290 BC00290 V=100.0  +MOVJ EC00290
SREFP 3 C00291 BC00291  +REFP EC00291
CALL JOB:SEARCH-R1-S13D
SET P044 P006
SFTON3D P044
SMOVL C00292 BC00292 V=133.3  +MOVJ EC00292
SMOVL C00293 BC00293 V=250.0  +MOVJ EC00293
SMOVL C00294 BC00294 V=133.3  +MOVJ EC00294
SREFP 3 C00295 BC00295  +REFP EC00295
CALL JOB:SEARCH-R1-S13D
SET P044 P006
SFTON3D P044
SMOVL C00296 BC00296 V=133.3  +MOVJ EC00296
SFTOF3D
MOVJ C00297 BC00297 VJ=30.00  +MOVJ EC00297 VJ=15.00
MOVJ C00298 BC00298 VJ=30.00  +MOVJ EC00298 VJ=15.00
MOVJ C00299 BC00299 VJ=30.00  +MOVJ EC00299 VJ=15.00
SMOVL C00300 BC00300 V=250.0  +MOVJ EC00300
SREFP 3 C00301 BC00301  +REFP EC00301
CALL JOB:SEARCH-R1-S13D
SET P045 P006
SFTON3D P045
SMOVL C00302 BC00302 V=250.0  +MOVJ EC00302
SREFP 3 C00303 BC00303  +REFP EC00303
CALL JOB:SEARCH-R1-S13D
SET P045 P006
SFTON3D P045
SMOVL C00304 BC00304 V=250.0  +MOVJ EC00304
SMOVL C00305 BC00305 V=250.0  +MOVJ EC00305
SMOVL C00306 BC00306 V=166.7  +MOVJ EC00306
SREFP 3 C00307 BC00307  +REFP EC00307
CALL JOB:SEARCH-R1-S13D
SET P045 P006
SFTON3D P045
SMOVL C00308 BC00308 V=250.0  +MOVJ EC00308
SFTOF3D
MOVJ C00309 BC00309 VJ=30.00  +MOVJ EC00309 VJ=15.00
MOVJ C00310 BC00310 VJ=30.00  +MOVJ EC00310 VJ=15.00
SMOVL C00311 BC00311 V=250.0  +MOVJ EC00311
SREFP 3 C00312 BC00312  +REFP EC00312
CALL JOB:SEARCH-R1-S13D
SET P046 P006
SFTON3D P046
SMOVL C00313 BC00313 V=250.0  +MOVJ EC00313
SREFP 3 C00314 BC00314  +REFP EC00314
CALL JOB:SEARCH-R1-S13D
SET P046 P006
SFTON3D P046
SMOVL C00315 BC00315 V=250.0  +MOVJ EC00315
SFTOF3D
MOVJ C00316 BC00316 VJ=30.00  +MOVJ EC00316 VJ=15.00
MOVJ C00317 BC00317 VJ=30.00  +MOVJ EC00317 VJ=15.00
MOVJ C00318 BC00318 VJ=30.00  +MOVJ EC00318 VJ=15.00
MOVJ C00319 BC00319 VJ=30.00  +MOVJ EC00319 VJ=15.00
SMOVL C00320 BC00320 V=250.0  +MOVJ EC00320
SREFP 3 C00321 BC00321  +REFP EC00321
CALL JOB:SEARCH-R1-S13D
SET P048 P006
SFTON3D P048
SMOVL C00322 BC00322 V=250.0  +MOVJ EC00322
SREFP 3 C00323 BC00323  +REFP EC00323
CALL JOB:SEARCH-R1-S13D
SET P048 P006
SFTON3D P048
SMOVL C00324 BC00324 V=250.0  +MOVJ EC00324
MOVJ C00325 BC00325 VJ=30.00  +MOVJ EC00325 VJ=15.00
SFTOF3D
MOVJ C00326 BC00326 VJ=30.00  +MOVJ EC00326 VJ=15.00
MOVJ C00327 BC00327 VJ=30.00  +MOVJ EC00327 VJ=15.00
SMOVL C00328 BC00328 V=166.7  +MOVJ EC00328
SREFP 3 C00329 BC00329  +REFP EC00329
CALL JOB:SEARCH-R1-S13D
SET P049 P006
SFTON3D P049
SMOVL C00330 BC00330 V=166.7  +MOVJ EC00330
SREFP 3 C00331 BC00331  +REFP EC00331
CALL JOB:SEARCH-R1-S13D
SET P049 P006
SFTON3D P049
SMOVL C00332 BC00332 V=166.7  +MOVJ EC00332
SMOVL C00333 BC00333 V=166.7  +MOVJ EC00333
SMOVL C00334 BC00334 V=166.7  +MOVJ EC00334
SREFP 3 C00335 BC00335  +REFP EC00335
CALL JOB:SEARCH-R1-S13D
SET P049 P006
SFTON3D P049
SMOVL C00336 BC00336 V=166.7  +MOVJ EC00336
SFTOF3D
MOVJ C00337 BC00337 VJ=30.00  +MOVJ EC00337 VJ=30.00
MOVJ C00338 BC00338 VJ=30.00  +MOVJ EC00338 VJ=30.00
MOVJ C00339 BC00339 VJ=30.00  +MOVJ EC00339 VJ=15.00
SMOVL C00340 BC00340 V=250.0  +MOVJ EC00340
SREFP 3 C00341 BC00341  +REFP EC00341
CALL JOB:SEARCH-R1-S13D
SET P050 P006
SFTON3D P050
SMOVL C00342 BC00342 V=250.0  +MOVJ EC00342
SREFP 3 C00343 BC00343  +REFP EC00343
CALL JOB:SEARCH-R1-S13D
SET P050 P006
SFTON3D P050
SMOVL C00344 BC00344 V=250.0  +MOVJ EC00344
SMOVL C00345 BC00345 V=250.0  +MOVJ EC00345
SMOVL C00346 BC00346 V=166.7  +MOVJ EC00346
SREFP 3 C00347 BC00347  +REFP EC00347
CALL JOB:SEARCH-R1-S13D
SET P050 P006
SFTON3D P050
SMOVL C00348 BC00348 V=166.7  +MOVJ EC00348
SFTOF3D
MOVJ C00349 BC00349 VJ=30.00  +MOVJ EC00349 VJ=15.00
MOVJ C00350 BC00350 VJ=30.00  +MOVJ EC00350 VJ=15.00
MOVJ C00351 BC00351 VJ=30.00  +MOVJ EC00351 VJ=15.00
MOVJ C00352 BC00352 VJ=30.00  +MOVJ EC00352 VJ=30.00
MOVJ C00353 BC00353 VJ=30.00  +MOVJ EC00353 VJ=30.00
MACRO1 MJ#(0) ARGF9
SFTON3D P042
SMOVL C00354 BC00354 V=166.7  +MOVJ EC00354
ARCON
SMOVC C00355 BC00355 V=8.3  +MOVJ EC00355
SMOVC C00356 BC00356 V=8.3  +MOVJ EC00356
SMOVC C00357 BC00357 V=8.3  +MOVJ EC00357
SMOVL C00358 BC00358 V=8.3  +MOVJ EC00358
ARCOF
SFTOF3D
SMOVL C00359 BC00359 V=250.0  +MOVJ EC00359
SMOVL C00360 BC00360 V=250.0  +MOVJ EC00360
SFTON3D P043
SMOVL C00361 BC00361 V=166.7  +MOVJ EC00361
ARCON
SMOVC C00362 BC00362 V=8.3  +MOVJ EC00362
SMOVC C00363 BC00363 V=8.3  +MOVJ EC00363
SMOVC C00364 BC00364 V=8.3  +MOVJ EC00364
SMOVL C00365 BC00365 V=8.3  +MOVJ EC00365
ARCOF
SFTOF3D
SMOVL C00366 BC00366 V=166.7  +MOVJ EC00366
SMOVL C00367 BC00367 V=250.0  +MOVJ EC00367
MOVJ C00368 BC00368 VJ=30.00  +MOVJ EC00368 VJ=30.00
MACRO1 MJ#(0) ARGF9
MOVJ C00369 BC00369 VJ=15.00  +MOVJ EC00369 VJ=10.00
SFTON3D P044
SMOVL C00370 BC00370 V=166.7  +MOVJ EC00370
ARCON
SMOVL C00371 BC00371 V=9.2  +MOVJ EC00371
SMOVL C00372 BC00372 V=9.2  +MOVJ EC00372
ARCOF
SFTOF3D
SMOVL C00373 BC00373 V=250.0  +MOVJ EC00373
SFTON3D P045
SMOVL C00374 BC00374 V=166.7  +MOVJ EC00374
ARCON
SMOVL C00375 BC00375 V=9.2  +MOVJ EC00375
SMOVL C00376 BC00376 V=9.2  +MOVJ EC00376
ARCOF
SMOVL C00377 BC00377 V=250.0  +MOVJ EC00377
SFTON3D P046
SMOVL C00378 BC00378 V=166.7  +MOVJ EC00378
ARCON
SMOVL C00379 BC00379 V=9.2  +MOVJ EC00379
SMOVL C00380 BC00380 V=9.2  +MOVJ EC00380
ARCOF
SFTOF3D
SMOVL C00381 BC00381 V=166.7  +MOVJ EC00381
SMOVL C00382 BC00382 V=250.0  +MOVJ EC00382
SMOVL C00383 BC00383 V=250.0  +MOVJ EC00383
SMOVL C00384 BC00384 V=250.0  +MOVJ EC00384
SFTON3D P045
SMOVL C00385 BC00385 V=166.7  +MOVJ EC00385
ARCON
SMOVL C00386 BC00386 V=10.0  +MOVJ EC00386
ARCOF
SMOVL C00387 BC00387 V=250.0  +MOVJ EC00387
SMOVL C00388 BC00388 V=333.3  +MOVJ EC00388
SFTON3D P044
SMOVL C00389 BC00389 V=166.7  +MOVJ EC00389
ARCON
SMOVL C00390 BC00390 V=10.0  +MOVJ EC00390
ARCOF
SMOVL C00391 BC00391 V=250.0  +MOVJ EC00391
MOVJ C00392 BC00392 VJ=20.00  +MOVJ EC00392 VJ=10.00
MOVJ C00393 BC00393 VJ=40.00  +MOVJ EC00393 VJ=10.00
MOVJ C00394 BC00394 VJ=20.00  +MOVJ EC00394 VJ=10.00
SFTON3D P050
SMOVL C00395 BC00395 V=166.7  +MOVJ EC00395
ARCON
SMOVL C00396 BC00396 V=9.2  +MOVJ EC00396
SMOVL C00397 BC00397 V=9.2  +MOVJ EC00397
ARCOF
SMOVL C00398 BC00398 V=166.7  +MOVJ EC00398
SFTON3D P049
SMOVL C00399 BC00399 V=166.7  +MOVJ EC00399
ARCON
SMOVL C00400 BC00400 V=9.2  +MOVJ EC00400
SMOVL C00401 BC00401 V=9.2  +MOVJ EC00401
SMOVL C00402 BC00402 V=9.2  +MOVJ EC00402
ARCOF
SMOVL C00403 BC00403 V=166.7  +MOVJ EC00403
SFTON3D P048
SMOVL C00404 BC00404 V=166.7  +MOVJ EC00404
ARCON
SMOVL C00405 BC00405 V=9.2  +MOVJ EC00405
SMOVL C00406 BC00406 V=9.2  +MOVJ EC00406
SMOVL C00407 BC00407 V=8.3  +MOVJ EC00407
ARCOF
SMOVL C00408 BC00408 V=166.7  +MOVJ EC00408
SMOVL C00409 BC00409 V=166.7  +MOVJ EC00409
SFTON3D P049
SMOVL C00410 BC00410 V=166.7  +MOVJ EC00410
ARCON
SMOVL C00411 BC00411 V=10.0  +MOVJ EC00411
ARCOF
SMOVL C00412 BC00412 V=250.0  +MOVJ EC00412
SFTON3D P050
SMOVL C00413 BC00413 V=200.0  +MOVJ EC00413
ARCON
SMOVL C00414 BC00414 V=10.0  +MOVJ EC00414
ARCOF
SFTOF3D
SMOVL C00415 BC00415 V=250.0  +MOVJ EC00415
MOVJ C00416 BC00416 VJ=60.00  +MOVJ EC00416 VJ=60.00
MOVJ C00417 BC00417 VJ=60.00  +MOVJ EC00417 VJ=60.00
MOVJ C00418 BC00418 VJ=60.00  +MOVJ EC00418 VJ=60.00
MOVJ C00419 BC00419 VJ=100.00  +MOVJ EC00419 VJ=100.00
END
